SUBAPPLICATION GreenWhiteBackground_Abscheider (* Subapplication Type *)
  (* Standard: 61499-2 *)
  (* Version 1.0, 2023-02-06, franz *)
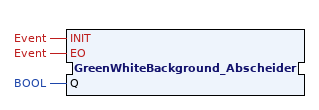
  EVENT_INPUT
    INIT;
    EO;
  END_EVENT
  VAR_INPUT
    Q : BOOL;
  END_VAR
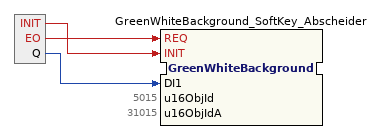
  FBS
    GreenWhiteBackground_SoftKey_Abscheider : GreenWhiteBackground(u16ObjId := 5015, u16ObjIdA := 31015);
  END_FBS
  EVENT_CONNECTIONS
    EO TO GreenWhiteBackground_SoftKey_Abscheider.REQ;
    INIT TO GreenWhiteBackground_SoftKey_Abscheider.INIT;
  END_CONNECTIONS
  DATA_CONNECTIONS
    Q TO GreenWhiteBackground_SoftKey_Abscheider.DI1;
  END_CONNECTIONS
END_SUBAPPLICATION
